// TIA Portal V20 export
DATA_BLOCK "SafetyCom_DB"   // DB45
// stored: AutoNumber false, InstanceOfName SafetyCom, InstanceOfType FB
"SafetyCom"
   // VAR
   //    Var { ExternalAccessible := 'False'; ExternalVisible := 'False'; ExternalWritable := 'False'} : "TypeVar";
   // END_VAR
BEGIN
END_DATA_BLOCK
